(* CoDeSys 2.3 export: MODBUS_TEST_HOLDING.EXP *)

(* POU PLC_PRG_mb, CFC *)
PROGRAM PLC_PRG_mb
VAR
	DD1: Read_Holding_Registers;					(*Блок опроса МВА*)
	DD2: R_TRIG;									(*Тригер, определяющий готовность блока*)
	DD3: MVA_Decode;								(*ФБ для расшифровки массива байт принятых по интерфейсу*)
	(*Входные данные*)
	DevAdr: BYTE := 16;								(*Адрес подключаемого прибора*)
	StartAdr: WORD := 0;							(*Адрес первого регистра для чтения*)
	Quantity: WORD := 48;							(*Число читаемых регистров*)
	DevNumb: WORD := 0;								(*Номер устройства Universal Network Modules*)
	t1:TIME:=T#150ms;								(*Максимальная задержка ответа*)
	t2:TIME:=T#50ms;								(*Пауза между запросами*)
	(*Результат*)
	Otvet: ARRAY [0..127] OF BYTE := 128(0);		(*Массив байт принятых от устройства*)
	ByteCount: WORD;								(*Число принятых байт*)
	Error: BYTE;									(*Ошибки*)
	Good_Count: WORD;								(*Число правильных запросов-ответов*)
	Error_Count: WORD;								(*Число не верных ответов-запросов*)
	MVA8: ARRAY [0..7] OF MVA8_AIN;					(*Массив структур - результат*)
	Errors: ARRAY [0..9] OF BYTE;					(*Массив ошибок*)
	e_count: BYTE;									(*Счетчик ошибок*)

	(*Вывод графика*)
	channel:BYTE:=3;								(*Номер выхода мва, выводимого на график*)
	t:REAL:=0;										(*Выводимое значение*)
END_VAR
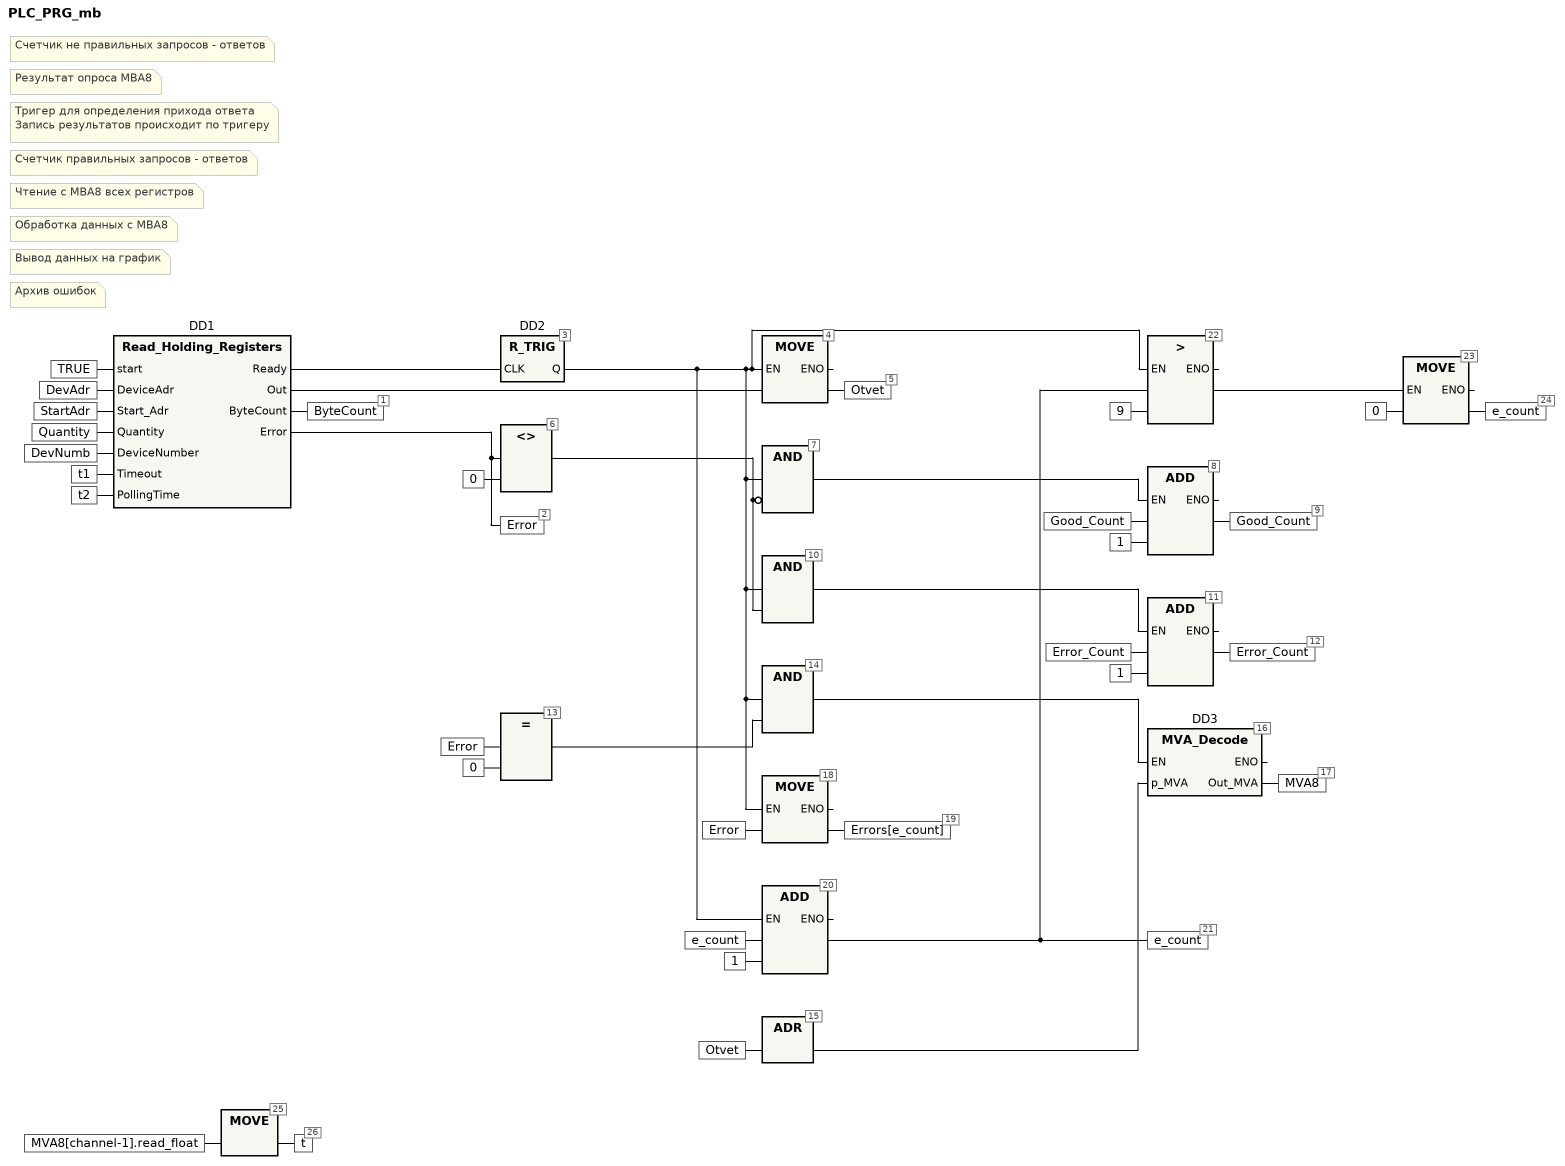
_CFC_ (* Continuous Function Chart, elements in execution order *)
(* Счетчик не правильных запросов - ответов *)
(* Результат опроса МВА8 *)
(* Тригер для определения прихода ответа / Запись результатов происходит по тригеру *)
(* Счетчик правильных запросов - ответов *)
(* Чтение с МВА8 всех регистров *)
(* Обработка данных с МВА8 *)
(* Вывод данных на график *)
#0 DD1:Read_Holding_Registers(start: TRUE, DeviceAdr: DevAdr, Start_Adr: StartAdr, Quantity: Quantity, DeviceNumber: DevNumb, Timeout: t1, PollingTime: t2)
#1 ByteCount <= #0.ByteCount
#2 Error <= #0.Error
(* Архив ошибок *)
#3 DD2:R_TRIG(CLK: #0.Ready)
#4 MOVE(EN: #3.Q, #0.Out)
#5 Otvet <= #4
#6 <>(#0.Error, 0)
#7 AND(#3.Q, NOT #6)
#8 ADD(EN: #7, Good_Count, 1)
#9 Good_Count <= #8
#10 AND(#3.Q, #6)
#11 ADD(EN: #10, Error_Count, 1)
#12 Error_Count <= #11
#13 =(Error, 0)
#14 AND(#3.Q, #13)
#15 ADR(Otvet)
#16 DD3:MVA_Decode(EN: #14, p_MVA: #15)
#17 MVA8 <= #16.Out_MVA
#18 MOVE(EN: #3.Q, Error)
#19 Errors[e_count] <= #18
#20 ADD(EN: #3.Q, e_count, 1)
#21 e_count <= #20
#22 >(EN: #3.Q, #20, 9)
#23 MOVE(EN: #22, 0)
#24 e_count <= #23
#25 MOVE(MVA8[channel-1].read_float)
#26 t <= #25
_END_CFC_
END_PROGRAM

(* POU Read_Holding_Registers, ST *)
FUNCTION_BLOCK Read_Holding_Registers

VAR_INPUT
	start:BOOL;									(*Разрешение работы блока*)
	DeviceAdr: BYTE;							(*Адрес устройства*)
	Start_Adr: WORD;							(*Адрес регистра с которого должно начаться чтение данных*)
	Quantity: WORD;								(*Число регистров для чтения*)
	DeviceNumber: WORD;							(*Адрес устройсва Universal Netvork Modul - начинаются с 0 сверху вниз*)
	Timeout:TIME;								(*Время ожидания ответа*)
	PollingTime:TIME;							(*Время между запросами*)
END_VAR

VAR_OUTPUT
	Ready:BOOL;									(*Готовность ФБ, ответ получен, или сформирована ошибка*)
	Out: ARRAY [0..127] OF BYTE;				(*Массив принятых байт*)
	ByteCount:WORD:=0;							(*Число байт в ответе*)
	Error: BYTE;								(*Код ошибки*)
END_VAR

VAR
	command_len: WORD := 8;						(*Длина команды для отправки*)
	command: ARRAY [0..127] OF BYTE := 128(0);	(*Команда*)
	command_string: STRING(128):='';			(*Строка команды для отправки*)

	stat:BYTE:=0;								(*Статус работы блока*)

	otvet_RB: POINTER TO RBDATA;				(*Структура ответа*)
	otvet: ARRAY [0..127] OF BYTE := 128(0);	(*Ответ*)
	count:INT;									(*Число принятых байт*)
	otvet_len: WORD;							(*Ожидаемая длина ответа*)
	otvet_len_error:WORD;						(*Ожидаемая длина ответа при наличии ошибки*)
	t1: TON;									(*Таймер ожидания ответа*)
	t2: TON;									(*Таймер между запросами*)
	modbus_error:BOOL:=FALSE;					(*Флаг, говорящий о том, что устройство прислало ошибку*)

	p:POINTER TO BYTE;							(*Указатели*)
	p1: POINTER TO BYTE;

	CRC: WORD:=0;								(*Контрольная сумма*)
	crc1:BYTE:=0;
	crc2:BYTE:=0;

	i: INT:=0;
END_VAR
(* @TEXT_IMPLEMENTATION := 'ST' *)
(*Если модуль не запущен, то освобождаем устройство Universal Netvork Module*)
IF NOT(start) THEN
	ReleaseDevice(DeviceNumber);
	stat:=0;
	ready:=FALSE;
ELSE
(*Если модуль запущен, то работаем с портом*)
	CASE stat OF
	0: (*Выполняем захват устройства*)
		IF(LockDevice(DeviceNumber)=1) THEN
			stat:=1;
		ELSE
			stat:=0;
		END_IF
		(*Инициализация переменных*)
		count:=0;
		ready:=FALSE;
		modbus_error:=FALSE;


	1:	(*Формируем команду запроса*)

		(*Адрес устройства*)
		command[0]:=DeviceAdr;
		(*Номер функции чтения 03h*)
		command[1]:=3;
		(*Стартовый адрес регистра*)
		p:=ADR(Start_Adr);
		command[3]:=p^;
		p:=ADR(Start_Adr)+1;
		command[2]:=p^;
		(*Число читаемых регистров*)
		p:=ADR(Quantity);
		command[5]:=p^;
		p:=ADR(Quantity)+1;
		command[4]:=p^;
		(*Расчет CRC*)
		p:=ADR(command);
		CRC:=MB_CRC(p, command_len-2);
		(*Вставляем в команду CRC*)
		p:=ADR(CRC);
		command[6]:=p^;
		p:=ADR(CRC)+1;
		command[7]:=p^;

		(*Расчет размера ожидаемого ответа*)
		otvet_len:=1+1+1+2*Quantity+2;	(*1х Адрес,1х функция,1х число байт,массивданных,2х CRC *)
		otvet_len_error:=1+1+1+2;		(*1х Адрес,1х ошибка83h,1х исключение,2х CRC *)

		stat:=2;

	2:	(*Копируем команду в строку для работы с модулем SetByte *)
		FOR i:=0 TO command_len-1 DO
			p:=ADR(command)+i;
			p1:=ADR(command_string)+i;
			p1^:=p^;
		END_FOR

		stat:=3;

	3:	(*Отсылаем команду*)
		IF SetByte(DeviceNumber, command_string, command_len)=command_len THEN
			stat:=4;
		ELSE
			stat:=3;
		END_IF

	4:	(*Запуск таймера ожидания ответа*)
		t1(IN:=TRUE , PT:=timeout );
		t1;
		stat:=5;

	5:	(*Прием ответа*)
		t1;
		otvet_RB:=GetByte(DeviceNumber);
		(*Если получили новый байт, то собираем его в результат*)
		(*и ведем подсчет принятых байт*)
		IF otvet_RB>0 THEN
			p:=ADR(otvet)+count;
			p^:=otvet_RB^.data;
			count:=count+1;
		END_IF

		(*Если получили первый байт, проверяем адрес устройства*)
		IF count=1 AND otvet[0]<>DeviceAdr AND t1.Q=FALSE THEN
			error:=1;
			t1(IN:=FALSE);
			t1;
			stat:=6;
			ready:=TRUE;
		END_IF

		(*Если получили второй байт, то проверяем размер посылки*)
		(*Или проверяем код ошибки*)
		IF count=2  AND t1.Q=FALSE THEN
			IF otvet[1]<>16#03 AND otvet[1]<>16#83 THEN
				error:=2;
				t1(IN:=FALSE);
				t1;
				stat:=6;
				ready:=TRUE;
			ELSIF otvet[1]=16#83 THEN
				modbus_error:=TRUE;
			END_IF
		END_IF

		(*Если получили третий байт, то проверяем размер посылки*)
		IF count=3 AND  modbus_error=FALSE AND otvet[2]<>Quantity*2 AND t1.Q=FALSE THEN
			error:=3;
			t1(IN:=FALSE);
			t1;
			stat:=6;
			ready:=TRUE;
		END_IF

		(*Если в ответе был код ошибки, то в третьем байте читаем исключение*)
		IF count=3 AND modbus_error=TRUE  AND t1.Q=FALSE THEN
			IF otvet[2]=1 THEN
				error:=4;
			ELSIF otvet[2]=2 THEN
				error:=5;
			ELSIF otvet[2]=3 THEN
				error:=6;
			ELSIF otvet[2]=4 THEN
				error:=7;
			ELSE
				error:=8;
			END_IF
		END_IF

		(*Если полностью пришел ошибочный ответ за допустимое время, проверяем CRC*)
		IF count=otvet_len_error AND modbus_error=TRUE AND t1.Q=FALSE  THEN
			(*Расчет CRC*)
			p:=ADR(otvet);
			CRC:=MB_CRC(p, otvet_len_error-2);
			p:=ADR(CRC);
			crc1:=p^;
			p:=ADR(CRC)+1;
			crc2:=p^;
			(*Сверяем CRC*)
			IF crc1=otvet[otvet_len_error-2] AND crc2=otvet[otvet_len_error-1] THEN
				error:=error;
			ELSE
				error:=9;
			END_IF
			t1(IN:=FALSE);
			t1;
			stat:=6;
			ready:=TRUE;
			modbus_error:=FALSE;
		END_IF

		(*Если получен ответ за допустимое время ожидания, то проверяем CRC *)
		(*И формируем результат*)
		IF count=otvet_len  AND t1.Q=FALSE  THEN
			(*Расчет CRC*)
			p:=ADR(otvet);
			CRC:=MB_CRC(p, otvet_len-2);
			p:=ADR(CRC);
			crc1:=p^;
			p:=ADR(CRC)+1;
			crc2:=p^;
			(*Сверяем CRC*)
			IF crc1=otvet[otvet_len-2] AND crc2=otvet[otvet_len-1] THEN
				error:=0;
				(*Выдаем результат*)
				FOR i:=0 TO Quantity*2-1 DO
					out[i]:=otvet[3+i];
				END_FOR

				FOR i:=Quantity*2 TO 127 DO
					out[i]:=0;
				END_FOR
				(*Выдаем число байт в ответе*)
				ByteCount:=Quantity*2;
			ELSE
				error:=10;
			END_IF
			t1(IN:=FALSE);
			t1;
			stat:=6;
			ready:=TRUE;
		END_IF

		IF t1.IN AND t1.Q THEN
			error:=11;
			t1(IN:=FALSE);
			t1;
			stat:=6;
			ready:=TRUE;
		END_IF

	6:	(*Организуем паузу между запросами*)
		t2(IN:=TRUE , PT:=PollingTime );
		t2;
		stat:=7;

	7:	(*Если задержка выполнена,то переходим к новому циклу опроса*)
		t2;
		GetByte(DeviceNumber);
		IF t2.IN AND t2.Q THEN
			t2(IN:=FALSE);
			t2;
			stat:=0;
		END_IF

	END_CASE

END_IF
END_FUNCTION_BLOCK

(* POU MB_CRC, ST *)
FUNCTION MB_CRC : WORD
VAR_INPUT
	pData: POINTER TO BYTE;		(* указатель на блок данных *)
	Size: WORD;						(* размер блока  данных *)
END_VAR
VAR
	Cnt: BYTE;							(* счетчик битов *)
END_VAR
(* @TEXT_IMPLEMENTATION := 'ST' *)
(* Вычисление контрольной суммы кадра MODBUS RTU CRC *)
MB_CRC := 16#FFFF;
WHILE Size > 0 DO
	MB_CRC := MB_CRC XOR pData^;
	FOR Cnt := 0 TO 7 DO
		IF MB_CRC.0 = 0 THEN
			MB_CRC := SHR(MB_CRC, 1);
		ELSE
			MB_CRC := SHR(MB_CRC, 1) XOR 16#A001;
		END_IF
	END_FOR;
	pData := pData + 1;
	Size := Size - 1;
END_WHILE
END_FUNCTION

(* POU MVA_Decode, ST *)
FUNCTION_BLOCK MVA_Decode
VAR_INPUT
	p_MVA:POINTER TO ARRAY [0..95] OF BYTE;
END_VAR
VAR_OUTPUT
	Out_MVA: ARRAY [0..7] OF MVA8_AIN;
END_VAR
VAR
	i:WORD:=0;
	p:POINTER TO BYTE;
	p1:POINTER TO BYTE;
END_VAR
(* @TEXT_IMPLEMENTATION := 'ST' *)
FOR i:=0 TO 95 BY 12 DO
	(*Читаем Сдвиг*)
	p:=ADR(p_MVA^[i])+1;
	p1:=ADR(Out_MVA[i/12].dp);
	p1^:=p^;
	P1:=P1+1;
	P:=P-1;
	p1^:=p^;
	(*Читаем целое значение*)
	p:=ADR(p_MVA^[i+2])+1;
	p1:=ADR(Out_MVA[i/12].read_int);
	p1^:=p^;
	P1:=P1+1;
	P:=P-1;
	p1^:=p^;
	(*Читаем статус измерения*)
	p:=ADR(p_MVA^[i+4])+1;
	p1:=ADR(Out_MVA[i/12].Error_Code);
	p1^:=p^;
	p1:=P1+1;
	P:=P-1;
	p1^:=p^;
	(*Читаем циклическое время измерения*)
	p:=ADR(p_MVA^[i+6])+1;
	p1:=ADR(Out_MVA[i/12].cykle_time);
	p1^:=p^;
	P1:=P1+1;
	P:=P-1;
	p1^:=p^;
	(*Читаем значение с плавающей точкой*)
	p:=ADR(p_MVA^[i+8])+3;
	p1:=ADR(Out_MVA[i/12].read_float);
	p1^:=p^;
	P1:=P1+1;
	P:=P-1;
	p1^:=p^;
	p:=ADR(p_MVA^[i+8])+1;
	p1:=ADR(Out_MVA[i/12].read_float)+2;
	p1^:=p^;
	P1:=P1+1;
	P:=P-1;
	p1^:=p^;
END_FOR
END_FUNCTION_BLOCK
